TYPE ST_AXIS_SYNCHRONISATION :
STRUCT
END_STRUCT
END_TYPE

(* stored: Version 1.1.0.1, ProductVersion 3.1.4024.11
   DUT ST_AXIS_SYNCHRONISATION: Id {2a9d6372-1c3e-4f42-82a7-c451b390d9d0} *)
